{attribute 'linkalways'} 
{attribute 'no_explicit_call' := 'This FB is a CLASS and must be accessed using methods or properties'}
{attribute 'enable_dynamic_creation'}
FUNCTION_BLOCK _ETcVnPixelConnectivity EXTENDS EnumDatatypeBase
VAR
	localData : ETcVnPixelConnectivity;
	activeData : REFERENCE TO ETcVnPixelConnectivity;
	enumBaseDatatype : _DINT(localData);
END_VAR

METHOD PRIVATE AddLocalEnumeration
VAR_INPUT
	Enumeration : T_MAXSTRING;
	Value : ETcVnPixelConnectivity;
END_VAR
AddEnumeration(Enumeration, Value);
END_METHOD

PROPERTY PUBLIC Address : PVOID
GET
Address := ADR(activeData);
END_GET
END_PROPERTY

METHOD PUBLIC ClearReference
VAR_INPUT
END_VAR
activeData REF= localData;
SetBaseDatatypeReference();
END_METHOD

METHOD PUBLIC Clone : I_Datatype
VAR
    pClone : POINTER TO _ETcVnPixelConnectivity;
END_VAR
pClone := __NEW(_ETcVnPixelConnectivity(InitialValue := Value));
Clone := pClone^;
END_METHOD

METHOD FB_init : BOOL
VAR_INPUT
	bInitRetains : BOOL; // if TRUE, the retain variables are initialized (warm start / cold start)
	bInCopyCode : BOOL;  // if TRUE, the instance afterwards gets moved into the copy code (online change)
	InitialValue : ETcVnPixelConnectivity;
END_VAR
localData := InitialValue;
AddBaseDatatype(enumBaseDatatype);
ClearReference();

AddLocalEnumeration('TCVN_PC_4', ETcVnPixelConnectivity.TCVN_PC_4);
AddLocalEnumeration('TCVN_PC_8', ETcVnPixelConnectivity.TCVN_PC_8);
END_METHOD

PROPERTY PUBLIC Identifier : T_MAXSTRING
GET
Identifier := 'ETcVnPixelConnectivity';
END_GET
END_PROPERTY

METHOD IsEnumeratorValueEqual : BOOL
VAR_INPUT
	Enumerator : I_KeyValueForwardEnumerator;
END_VAR
VAR
	storedValue : ETcVnPixelConnectivity;
END_VAR
IF NOT Enumerator.TryGet(storedValue) THEN
	RETURN;
END_IF

IsEnumeratorValueEqual := storedValue = activeData;
END_METHOD

METHOD PUBLIC MakeReferenceTo
VAR_INPUT
	ReferenceTarget : REFERENCE TO ETcVnPixelConnectivity;
END_VAR
activeData REF= ReferenceTarget;
SetBaseDatatypeReference();
END_METHOD

METHOD PROTECTED SetBaseDatatypeReference
VAR_INPUT
END_VAR
enumBaseDatatype.MakeReferenceTo(activeData);
END_METHOD

PROPERTY PUBLIC Size : UDINT
GET
Size := SIZEOF(activeData);
END_GET
END_PROPERTY

METHOD TryMakeReferenceTo : BOOL
VAR_INPUT
	Target : I_Datatype;
END_VAR
VAR
	targetAsEnum : I_EnumDatatype;
	pTargetData : POINTER TO ETcVnPixelConnectivity;
END_VAR
IF NOT Target.TryResolveAsEnumDatatype(targetAsEnum) THEN
	RETURN;
END_IF

IF targetAsEnum.Identifier <> Identifier THEN
	RETURN;
END_IF

pTargetData := Target.Address;
activeData REF= pTargetData^;
SetBaseDatatypeReference();
TryMakeReferenceTo := TRUE;
END_METHOD

PROPERTY PUBLIC Value : ETcVnPixelConnectivity
GET
Value := activeData;
END_GET
SET
activeData := Value;
END_SET
END_PROPERTY

END_FUNCTION_BLOCK

(* stored: Version 1.1.0.1
   POU _ETcVnPixelConnectivity: Id {bbd4df20-6c65-453c-964d-327271d928f1}, SpecialFunc None
   Folder Constructor: Id {9b8c0d72-1aff-4ace-92e7-616f65b4f591}
   Folder Private: Id {cf7b968d-9a01-49ef-9dcd-9f42be07cbba}
   Folder Protected: Id {35ed32fb-a95b-4389-a264-e697a654c0fa}
   Method AddLocalEnumeration: Id {da19d6cf-52e0-4a6f-bd3d-bd6d16330f8a}
   Property Address: Id {2f5f7f76-3a25-4dfc-bece-3cdb3f020c1a}
   Get Get: Id {54d26d0e-101c-4c69-aa8b-941cd690a87d}
   Method ClearReference: Id {17fbd375-13c4-438e-b660-3f9a6d21c8c4}
   Method Clone: Id {97d6ed79-f76b-4d6a-81e0-eec7c079b402}
   Method FB_init: Id {ca873e15-2126-46ed-ab46-d32c56c817c4}
   Property Identifier: Id {8f792aee-edda-4dca-9851-d393a109afc3}
   Get Get: Id {2a4154b9-af06-46ed-b7ae-369b990e6174}
   Method IsEnumeratorValueEqual: Id {3cc915e4-07d3-494b-8f03-7b25ae7930b4}
   Method MakeReferenceTo: Id {9f61669c-05cf-4ab7-bed1-0794483ac9e8}
   Method SetBaseDatatypeReference: Id {735173c9-e107-4bcc-a051-eddc146cb253}
   Property Size: Id {4b9a8ce3-b2f0-4875-be7f-a382c4c06c05}
   Get Get: Id {03e69c60-1204-46a2-bf91-2f6af0b9fd64}
   Method TryMakeReferenceTo: Id {d205c2d9-b1cb-4b0a-89d3-242ff5cf81b4}
   Property Value: Id {caf35543-fbf1-44bf-b241-f4cc14e78b7c}
   Get Get: Id {6e6c75d5-1f58-425d-bfb6-f2bada463f78}
   Set Set: Id {b3e2eb1f-f791-422f-ac17-dde696e7a3c8} *)
